FUNCTION_BLOCK fbSignalSimSlider
VAR_IN_OUT
	em : ST_EM;
END_VAR
VAR_INPUT
	EnableSim : BOOL;
	UnknownStartPosition : BOOL := FALSE;
	StartOnOtherSide : BOOL := FALSE;
END_VAR
VAR
	InitialConfig : BOOL := TRUE;
	timers : ARRAY[1..10] OF TON;
	duration : TIME := T#5S;
	elapsed : TIME;
	OtherSide : BOOL := FALSE;
END_VAR

IF EnableSim THEN
	IF InitialConfig THEN
		InitialConfig := FALSE;
		IF NOT UnknownStartPosition THEN
			IF StartOnOtherSide THEN
				em.Config.Data.I[2] := TRUE;
				OtherSide := TRUE;
			ELSE
				em.Config.Data.I[1] := TRUE;
			END_IF
		ELSE
			em.Config.Data.I[1] := FALSE;
			em.Config.Data.I[2] := FALSE;
		END_IF
	END_IF
	
	timers[1].PT := timers[2].PT := timers[3].PT := timers[10].PT := duration;
	timers[4].PT := timers[5].PT := timers[6].PT := timers[7].PT := timers[8].PT := timers[9].PT := duration / 3;
	
	CASE em.SequenceStep OF
		10:	timers[5](in := TRUE);
		
			IF timers[5].Q THEN
				timers[5](in := FALSE);
				em.Cmd := E_CMD.clear;
			END_IF 
	
		30:	timers[6](in := TRUE);
		
			IF timers[6].Q THEN
				timers[6](in := FALSE);
				em.Cmd := E_CMD.reset;	
			END_IF

		35:	timers[10](in := TRUE);
		
			IF timers[10].Q THEN
				timers[10](in := FALSE);
				em.Config.Data.I[1] := TRUE;
			END_IF
	
		40: timers[4](in := TRUE);
		
			IF timers[4].Q THEN
				timers[4](in := FALSE);
				em.Cmd := E_CMD.start;
			END_IF	

		50:	IF NOT OtherSide AND em.Config.Data.I[1] THEN
				timers[1](in := TRUE); 
			END_IF
			
			IF timers[1].Q THEN
				timers[1](in := FALSE);
				em.Config.Data.I[3] := TRUE;
			END_IF
			
		60:	IF NOT OtherSide AND em.Config.Data.I[1] THEN
				timers[2](in := NOT timers[2].Q);
			ELSE
				timers[3](in := NOT timers[3].Q);
			END_IF
			
			em.Config.Data.I[1] := FALSE;
			em.Config.Data.I[2] := FALSE;
			em.Config.Data.I[3] := FALSE;
			
			IF timers[2].Q THEN
				timers[2](in := FALSE);
				em.Config.Data.I[2] := TRUE;
			END_IF
			
			IF timers[3].Q THEN
				timers[3](in := FALSE);
				em.Config.Data.I[1] := TRUE;
			END_IF
			
		200:timers[8](in := TRUE);
		
			IF timers[8].Q THEN
				timers[8](in := FALSE);
				em.Cmd := E_CMD.unhold;	
			END_IF
		
		300:timers[9](in := TRUE);
		
			IF timers[9].Q THEN
				timers[9](in := FALSE);
				em.Cmd := E_CMD.unsuspend;	
			END_IF
	END_CASE

	OtherSide := FALSE;
END_IF

END_FUNCTION_BLOCK

(* stored: Version 1.1.0.1, ProductVersion 3.1.4024.12
   POU fbSignalSimSlider: Id {c8e777ba-6f9f-4e87-b459-2b373f0a1647}, SpecialFunc None *)
